Omron CX-Programmer project NewProject (CX-Programmer 9.75)

# PLC NewPLC1: CP1H XA

## Global symbols (name address type ; comment)
0.00 BOOL  ; PB1
0.01 BOOL  ; STOP
0.02 BOOL  ; SENSOR1
0.03 BOOL  ; RESET1
0.04 BOOL  ; PB2
0.05 BOOL  ; SENSOR3
0.06 BOOL  ; RESET2
100.00 BOOL  ; CONTACTOR1
101.00 BOOL  ; CONVEYOR1
102.00 BOOL  ; FILLING
103.00 BOOL  ; CAPPING
104.00 BOOL  ; MOVING
105.00 BOOL  ; CONTACTOR2
106.00 BOOL  ; CONVEYOR2
107.00 BOOL  ; PACKING
C0000 BOOL  ; Count
C0001 BOOL  ; BOTTLE COUNT
C0002 BOOL  ; BOTTLE COUNT2
T0001 BOOL  ; TIME1
T0002 BOOL  ; TIME2
T0003 BOOL  ; TIME3
T0004 BOOL  ; TIME4
T0005 BOOL  ; TIME5
T0006 BOOL  ; TIME6
T0007 BOOL  ; TIME7

## Program NewProgram1 (cyclic task 0)

### Section Section1

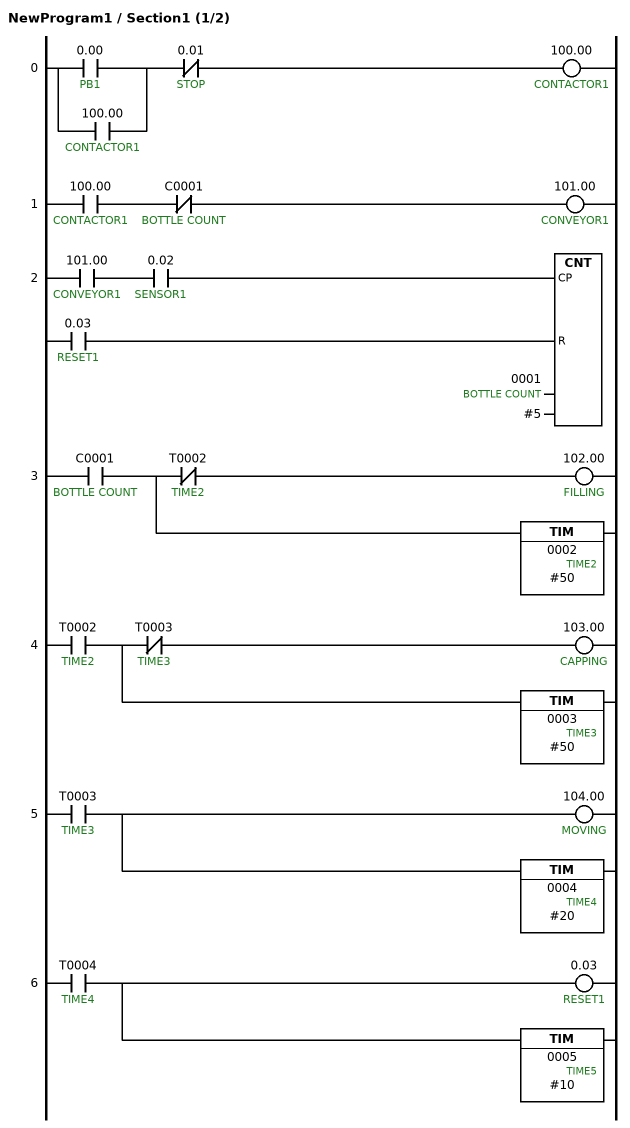
; rung 0
LD 0.00  ; PB1
OR 100.00  ; CONTACTOR1
ANDNOT 0.01  ; STOP
OUT 100.00  ; CONTACTOR1
; rung 1
LD 100.00  ; CONTACTOR1
ANDNOT C0001  ; BOTTLE COUNT
OUT 101.00  ; CONVEYOR1
; rung 2
LD 101.00  ; CONVEYOR1
AND 0.02  ; SENSOR1
LD 0.03  ; RESET1
CNT 0001 #5  ; BOTTLE COUNT
; rung 3
LD C0001  ; BOTTLE COUNT
OUT TR0
ANDNOT T0002  ; TIME2
OUT 102.00  ; FILLING
LD TR0
TIM 0002 #50  ; TIME2
; rung 4
LD T0002  ; TIME2
OUT TR0
ANDNOT T0003  ; TIME3
OUT 103.00  ; CAPPING
LD TR0
TIM 0003 #50  ; TIME3
; rung 5
LD T0003  ; TIME3
OUT 104.00  ; MOVING
TIM 0004 #20  ; TIME4
; rung 6
LD T0004  ; TIME4
OUT 0.03  ; RESET1
TIM 0005 #10  ; TIME5

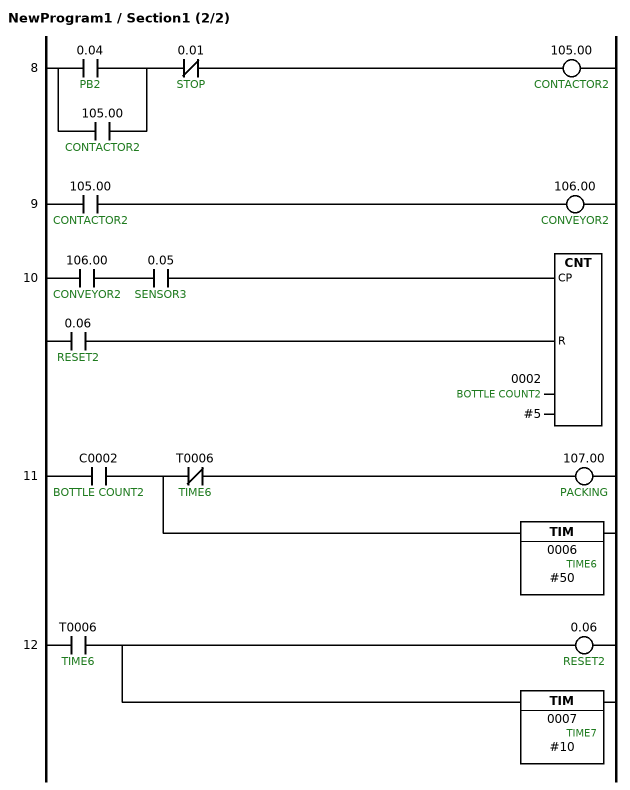
; rung 8
LD 0.04  ; PB2
OR 105.00  ; CONTACTOR2
ANDNOT 0.01  ; STOP
OUT 105.00  ; CONTACTOR2
; rung 9
LD 105.00  ; CONTACTOR2
OUT 106.00  ; CONVEYOR2
; rung 10
LD 106.00  ; CONVEYOR2
AND 0.05  ; SENSOR3
LD 0.06  ; RESET2
CNT 0002 #5  ; BOTTLE COUNT2
; rung 11
LD C0002  ; BOTTLE COUNT2
OUT TR0
ANDNOT T0006  ; TIME6
OUT 107.00  ; PACKING
LD TR0
TIM 0006 #50  ; TIME6
; rung 12
LD T0006  ; TIME6
OUT 0.06  ; RESET2
TIM 0007 #10  ; TIME7

### Section END
; rung 0
END(001)